{attribute 'GeneratedUsingTerminal: EJ2521-0224-0016'}
{attribute addProperty BoxType "EJ2521-0224-0016"}
{attribute addProperty Id "ControlAT %Q*Control_7786EF9F2Switch_on_valueAT %Q*UINT2Switch_off_valueAT %Q*UINT2"}
{attribute addProperty CRC "3446555870"}
{attribute addProperty Size "6"}
TYPE PLS_Control_compact_Channel_CD6E44DE :
STRUCT
	{attribute addProperty Name "Control"}
	Control AT %Q* : Control_7786EF9F;
	{attribute addProperty Name "Switch_on_value"}
	Switch_on_value AT %Q* : UINT;
	{attribute addProperty Name "Switch_off_value"}
	Switch_off_value AT %Q* : UINT;
END_STRUCT
END_TYPE

(* stored: Version 1.2.0.0, ProductVersion 3.1.4024.9
   DUT PLS_Control_compact_Channel_CD6E44DE: Id {792addb3-89ab-44ec-a830-8dba47daa77a} *)
